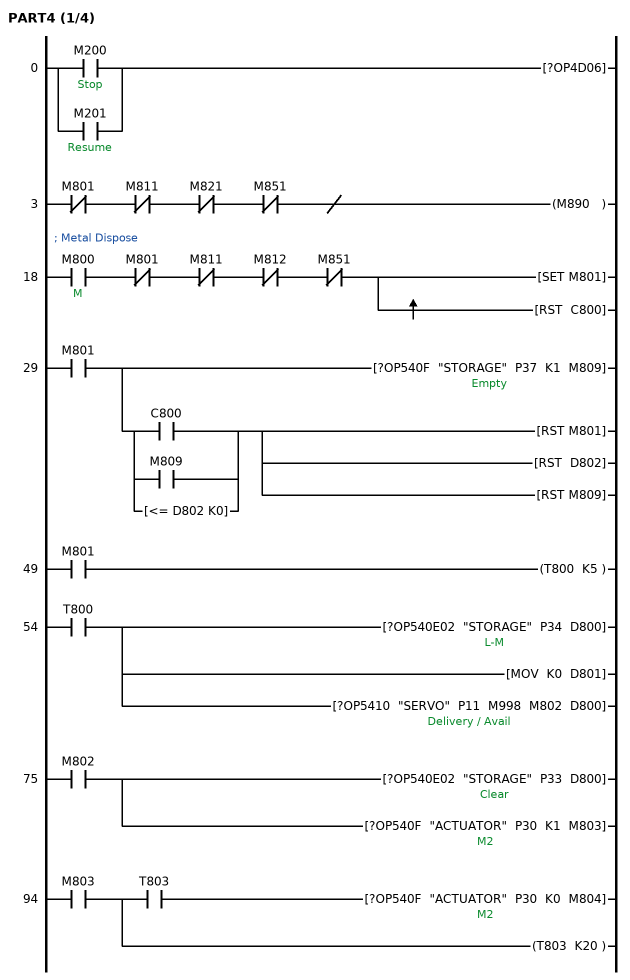
[picture p24: ladder of PART4, rungs at steps 0 to 94]
0     LD      M200  ; Stop
      OR      M201  ; Resume
      ?OP4D06
3     LDI     M801
      ANI     M811
      ANI     M821
      ANI     M851
      INV
      OUT     M890
; Metal Dispose
18    LD      M800  ; M
      ANI     M801
      ANI     M811
      ANI     M812
      ANI     M851
      SET     M801
      MEP
      RST     C800
29    LD      M801
      ?OP540F "STORAGE" P37 K1 M809  ; Empty
      LD      C800
      OR      M809
      OR<=    D802 K0
      ANB
      RST     M801
      RST     D802
      RST     M809
49    LD      M801
      OUT     T800 K5
54    LD      T800
      ?OP540E02 "STORAGE" P34 D800  ; L-M
      MOV     K0 D801
      ?OP5410 "SERVO" P11 M998 M802 D800  ; Delivery / Avail
75    LD      M802
      ?OP540E02 "STORAGE" P33 D800  ; Clear
      ?OP540F "ACTUATOR" P30 K1 M803  ; M2
94    LD      M803
      MPS
      AND     T803
      ?OP540F "ACTUATOR" P30 K0 M804
      MPP
      OUT     T803 K20
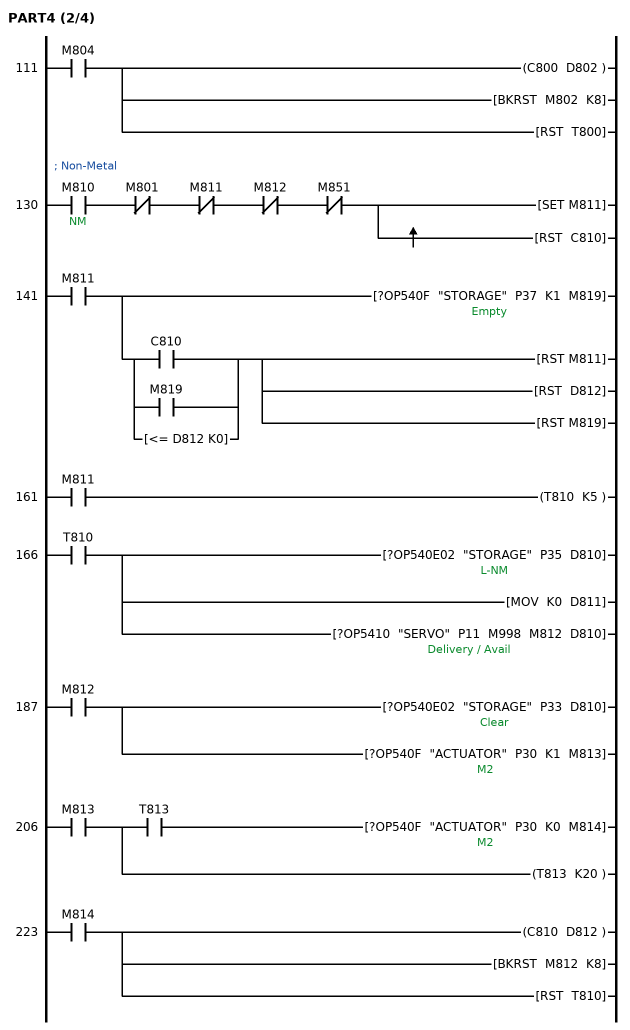
111   LD      M804
      OUT     C800 D802
      BKRST   M802 K8
      RST     T800
; Non-Metal
130   LD      M810  ; NM
      ANI     M801
      ANI     M811
      ANI     M812
      ANI     M851
      SET     M811
      MEP
      RST     C810
141   LD      M811
      ?OP540F "STORAGE" P37 K1 M819
      LD      C810
      OR      M819
      OR<=    D812 K0
      ANB
      RST     M811
      RST     D812
      RST     M819
161   LD      M811
      OUT     T810 K5
166   LD      T810
      ?OP540E02 "STORAGE" P35 D810  ; L-NM
      MOV     K0 D811
      ?OP5410 "SERVO" P11 M998 M812 D810
187   LD      M812
      ?OP540E02 "STORAGE" P33 D810
      ?OP540F "ACTUATOR" P30 K1 M813
206   LD      M813
      MPS
      AND     T813
      ?OP540F "ACTUATOR" P30 K0 M814
      MPP
      OUT     T813 K20
223   LD      M814
      OUT     C810 D812
      BKRST   M812 K8
      RST     T810
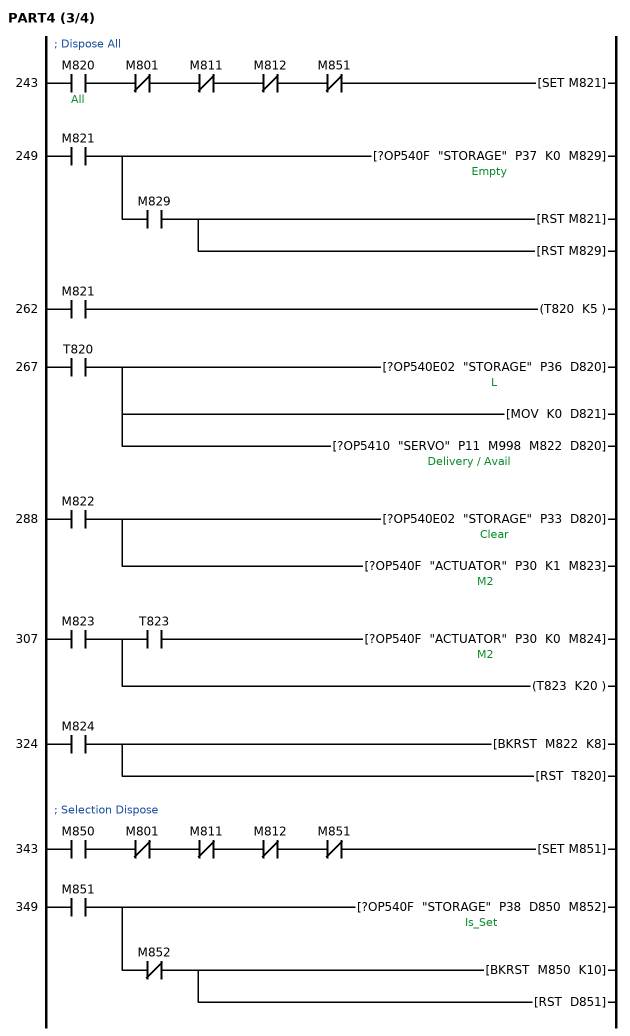
; Dispose All
243   LD      M820  ; All
      ANI     M801
      ANI     M811
      ANI     M812
      ANI     M851
      SET     M821
249   LD      M821
      ?OP540F "STORAGE" P37 K0 M829
      AND     M829
      RST     M821
      RST     M829
262   LD      M821
      OUT     T820 K5
267   LD      T820
      ?OP540E02 "STORAGE" P36 D820  ; L
      MOV     K0 D821
      ?OP5410 "SERVO" P11 M998 M822 D820
288   LD      M822
      ?OP540E02 "STORAGE" P33 D820
      ?OP540F "ACTUATOR" P30 K1 M823
307   LD      M823
      MPS
      AND     T823
      ?OP540F "ACTUATOR" P30 K0 M824
      MPP
      OUT     T823 K20
324   LD      M824
      BKRST   M822 K8
      RST     T820
; Selection Dispose
343   LD      M850
      ANI     M801
      ANI     M811
      ANI     M812
      ANI     M851
      SET     M851
349   LD      M851
      ?OP540F "STORAGE" P38 D850 M852  ; Is_Set
      ANI     M852
      BKRST   M850 K10
      RST     D851
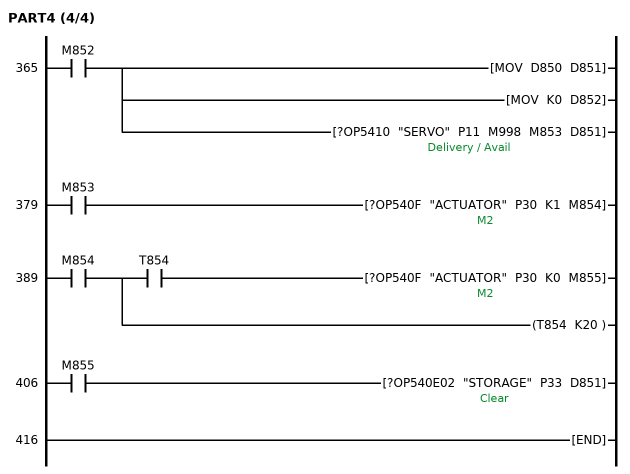
365   LD      M852
      MOV     D850 D851
      MOV     K0 D852
      ?OP5410 "SERVO" P11 M998 M853 D851
379   LD      M853
      ?OP540F "ACTUATOR" P30 K1 M854
389   LD      M854
      MPS
      AND     T854
      ?OP540F "ACTUATOR" P30 K0 M855
      MPP
      OUT     T854 K20
406   LD      M855
      ?OP540E02 "STORAGE" P33 D851
416   END
END_PROGRAM

PROGRAM LAMP1
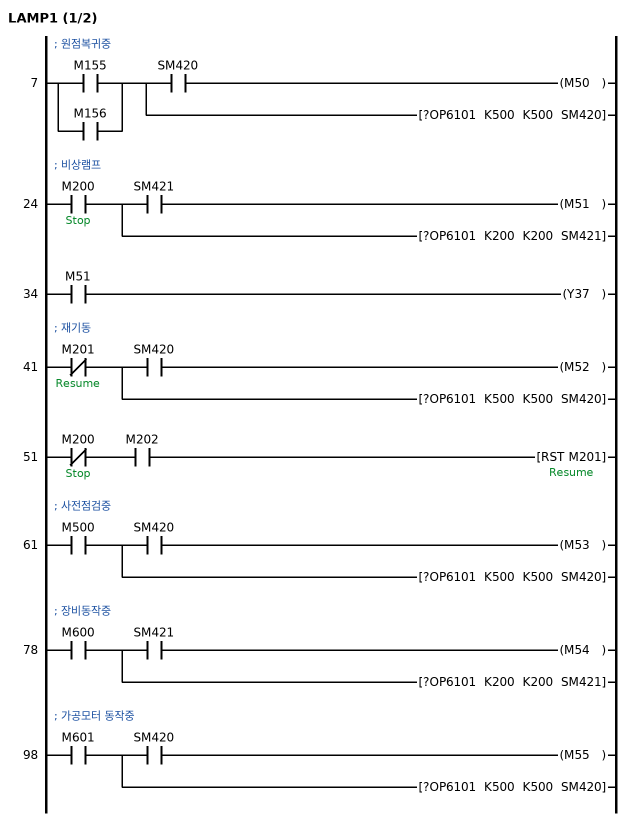
; 원점복귀중
7     LD      M155
      OR      M156
      MPS
      AND     SM420
      OUT     M50
      MPP
      ?OP6101 K500 K500 SM420
; 비상램프
24    LD      M200  ; Stop
      MPS
      AND     SM421
      OUT     M51
      MPP
      ?OP6101 K200 K200 SM421
34    LD      M51
      OUT     Y37
; 재기동
41    LDI     M201  ; Resume
      MPS
      AND     SM420
      OUT     M52
      MPP
      ?OP6101 K500 K500 SM420
51    LDI     M200  ; Stop
      AND     M202
      RST     M201  ; Resume
; 사전점검중
61    LD      M500
      MPS
      AND     SM420
      OUT     M53
      MPP
      ?OP6101 K500 K500 SM420
; 장비동작중
78    LD      M600
      MPS
      AND     SM421
      OUT     M54
      MPP
      ?OP6101 K200 K200 SM421
; 가공모터 동작중
98    LD      M601
      MPS
      AND     SM420
      OUT     M55
      MPP
      ?OP6101 K500 K500 SM420
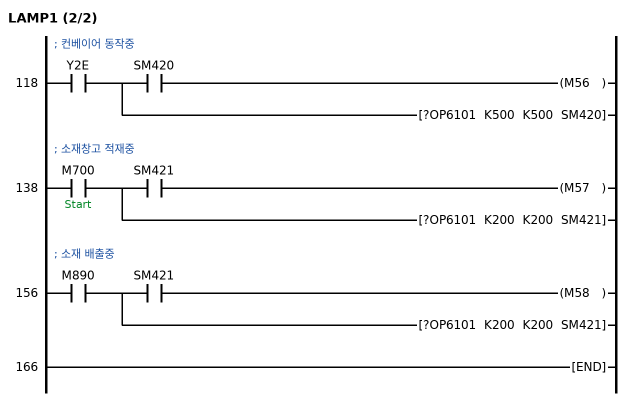
; 컨베이어 동작중
118   LD      Y2E
      MPS
      AND     SM420
      OUT     M56
      MPP
      ?OP6101 K500 K500 SM420
; 소재창고 적재중
138   LD      M700  ; Start
      MPS
      AND     SM421
      OUT     M57
      MPP
      ?OP6101 K200 K200 SM421
; 소재 배출중
156   LD      M890
      MPS
      AND     SM421
      OUT     M58
      MPP
      ?OP6101 K200 K200 SM421
166   END
END_PROGRAM

// device comments not shown above
P0  ; Open
P1  ; Wait
P2  ; Delivery
P3  ; Move
P6  ; F-Return
P16  ; F-Return
P20  ; Reset
P51  ; Set
M220  ; A+
M221  ; A-
M996  ; Stop
D330  ; Set
D341  ; Latest
D351  ; Latest
R0  ; Cnt
R1  ; Set Bits
R2  ; M
R3  ; NM
